PROGRAM prg_ADS
VAR
	ADS_1: FB_ADS_Read;
	str_ADS_read: STRING(40);
	byte_array : ARRAY[0..1023] OF BYTE;
	struct_received	: struct_ADS_Reichinger;						
	
	int_liveCount		: INT;						//{#lynus.ag#()}
	byte_old: BYTE;
	m_ADS_Error: BOOL;								//{#lynus.ag#()}
	int_ADS_Received_Count: INT;					//{#lynus.ag#()}
END_VAR


str_ADS_read := 'prgLynusCom.byte_array';

ADS_1(
	udintWriteLength:=  SIZEOF(byte_array), 
	udintReadLength:= SIZEOF(byte_array), 
	dwSourceAddr:= ADR(str_ADS_read), 
	dwDestAddr:= ADR(byte_array), 
	strNetID:= '5.100.32.101.1.1', 
	timeReadDelay:= T#5S, 
	mADSError=> , 
	strADSErrorText=> );
	
// copy struct to byte array
IF byte_array[1] <> byte_old AND NOT ADS_1.mADSError AND byte_array[1] <> 0 THEN
	IF SIZEOF(struct_received) > SIZEOF(byte_array) THEN
		memcpy(ADR(struct_received),ADR(byte_array),SIZEOF(byte_array));
	ELSE
		memcpy(ADR(struct_received),ADR(byte_array),SIZEOF(struct_received));
	END_IF
	byte_old := byte_array[1];
	int_ADS_Received_Count := int_ADS_Received_Count+1;
END_IF
m_ADS_Error := ADS_1.mADSError;
	
	
int_liveCount := struct_received.int_liveCount;

END_PROGRAM

(* stored: Version 1.1.0.1, ProductVersion 3.1.4024.12
   POU prg_ADS: Id {1ec2d5ec-bf1c-4c74-8834-68e6bec7f66c}, SpecialFunc None *)
